// TIA Portal V17 export
// export: Created 2023-02-14T02:49:13.374169Z, ExportSetting WithDefaults, DisplayName Totally Integrated Automation Portal, DisplayVersion V17, DisplayName TIA Portal Openness, DisplayVersion V17, DisplayName TIA Portal Teamcenter Gateway, DisplayVersion V17, DisplayName TIA Portal Version Control Interface, DisplayVersion V17, DisplayName SINAMICS Startdrive Advanced, DisplayVersion V17, DisplayName SINAMICS Startdrive G130, G150, S120, S150, SINAMICS MV, S210, DisplayVersion V17, DisplayName SINAMICS Startdrive G110M, G120, G120C, G120D, G120P, G115D, DisplayVersion V17, DisplayName STEP 7 Professional, DisplayVersion V17, DisplayName STEP 7 Safety, DisplayVersion V17, DisplayName WinCC Professional, DisplayVersion V17
DATA_BLOCK "Salt_to_Mix"   // DB21
{ S7_Optimized_Access := 'FALSE' }
VERSION : 0.1
// stored: AutoNumber true, DBAccessibleFromOPCUA true, DBAccessibleFromWebserver true, IsOnlyStoredInLoadMemory false, IsWriteProtectedInAS false
   VAR
      Heartbeat : Bool;   // Alternating value of 0 and 1 to indicate that the PLC is alive
      "System ready to run" : Bool;   // Gericke system is ready to receive signal from customer
      "Batching in process" : Bool;   // Signal received from customer, system is in batching process
      "Batching on hold" : Bool;   // Batching process on hold (either by alarm or manual hold by operator)
      "Batching completed" : Bool;   // Batching process completed, system will proceed to PTA transfer
      "Batching alarm" : Bool;   // Batching alarm exist (tolerance alarm, loadcell fault, etc)
      "PTA in process" : Bool;   // PTA transfer in process
      "PTA completed" : Bool;   // PTA transfer completed
      "PTA warning alarm" : Bool;   // PTA warning alarm exist (Conveying timeout, Filling timeout, etc)
      "PTA critical alarm" : Bool;   // Alarm exist (Overpressure, etc)
   END_VAR
BEGIN
END_DATA_BLOCK
